PROGRAM MAIN
VAR
	floorOneLamp : BOOL := FALSE;
END_VAR


CheckIfAtFloor();

CASE GVL.caseInput OF
	0:
		// Init lift values
		GVL.currentFloor := 0;
		GVL.targetFloor := 0;
		GVL.liftMoving := FALSE;
		GVL.openDoor := FALSE;
		
		// Set lift to operating mode
		GVL.caseInput := 1;

	1:
		// Wait for outside user input
		IF GVL.callLevel0 THEN
			GVL.targetFloor := 0;
			GVL.ledLevel0 := TRUE;
			// Set the case input
			GVL.caseInput := 2;
		ELSIF GVL.callLevel1 THEN
			GVL.targetFloor := 1;
			GVL.ledLevel1 := TRUE;
			// Set the case input
			GVL.caseInput := 2;
		ELSIF GVL.callLevel2 THEN
			GVL.targetFloor := 2;
			GVL.ledLevel2 := TRUE;
			// Set the case input
			GVL.caseInput := 2;
		END_IF
			
	2:
		// Check if at target floor
		IF GVL.targetFloor = GVL.currentFloor THEN
			// Stop lift movements
			GVL.liftMoving := FALSE;
			
			// Turn off ledLevels
			GVL.ledLevel0 := FALSE;
			GVL.ledLevel1 := FALSE;
			GVL.ledLevel2 := FALSE;
			
			// Open the door
			GVL.openDoor := TRUE;
			
			// Set case to 5 and wait for user input
			GVL.caseInput := 5;
			
		ELSIF GVL.targetFloor < GVL.currentFloor THEN
			GVL.caseInput := 3;
		ELSIF GVL.targetFloor > GVL.currentFloor THEN
			GVL.caseInput := 4;
		END_IF
		
	3:
		// Move lift upwards
		GVL.liftDirection := TRUE;
		GVL.liftMoving := TRUE;
		
		// SInulate lift timer
		GVL.simulationTime(IN := TRUE, PT := GVL.simulationPace);
		
		// Increase lift level by 1
		GVL.currentFloor := GVL.currentFloor + 1;
		
		// Check if this is the correct floor
		GVL.caseInput := 2;
		
	4: // Move lift downwards
		GVL.liftDirection := FALSE;
		GVL.liftMoving := TRUE;
		
		// SInulate lift timer
		GVL.simulationTime(IN := TRUE, PT := GVL.simulationPace);
		
		// Decrease lift level by 1
		GVL.currentFloor := GVL.currentFloor - 1;
		
		// Check if this is the correct floor
		GVL.caseInput := 2;
		
	5:
		// Wait for user input inside lift to move
		IF GVL.setTargetLevel0 THEN
			GVL.targetFloor := 0;
			GVL.caseInput := 2;
		ELSIF GVL.setTargetLevel1 THEN
			GVL.targetFloor := 1;
			GVL.caseInput := 2;
		ELSIF GVL.setTargetLevel2 THEN
			GVL.targetFloor := 2;
			GVL.caseInput := 2;
		END_IF
		
END_CASE

END_PROGRAM

(* stored: Version 1.1.0.1, ProductVersion 3.1.4024.12
   POU MAIN: Id {691ad225-5b7f-4f82-b1a8-a7e9bbc42919}, SpecialFunc None *)
